// TIA Portal V20 export
// export: Created 2025-12-01T14:56:19.1379541Z, ExportSetting None, DisplayName Totally Integrated Automation Portal, DisplayVersion V20 Update 3, DisplayName TIA Portal Openness, DisplayVersion V20 Update 3, DisplayName TIA Portal Version Control Interface, DisplayVersion V20 Update 3, DisplayName STEP 7 Professional, DisplayVersion V20 Update 3, DisplayName STEP 7 Safety, DisplayVersion V20 Update 2, DisplayName WinCC Basic/Comfort/Advanced, DisplayVersion V20 Update 3, DisplayName WinCC Professional, DisplayVersion V20 Update 3, DisplayName WinCC Unified, DisplayVersion V20 Update 3
TYPE "i550 Estatus variador"
   STRUCT
      "Digital input 1" : Bool;   // DI1 Entrada digital 1 xxxx.0
      "Digital input 2" : Bool;   // DI2 Entrada digital 2 xxxx.1
      "Digital input 3" : Bool;   // DI3 Entrada digital 3 xxxx.2
      "Digital input 4" : Bool;   // DI4 Entrada digital 4 xxxx.3
      "Digital input 5" : Bool;   // DI5 Entrada digital 5 xxxx.4
      Running : Bool;
      "Release Holding Brake" : Bool;
      "Reserva 3" : Bool;
      "Ready for operation" : Bool;   // Dispositivo OK para su utilización
      "Auto setp active" : Bool;   // Modo auto activo
      "Actual speed = 0" : Bool;   // Velocidad actual = 0
      Error : Bool;   // Dispositivo en error
      "Safe torque off" : Bool;   // STO no activo en dispositivo
      "At current limit" : Bool;   // Corriente limite superada
      "At torque limit" : Bool;   // Par limite superado
      "Speed - set = act" : Bool;   // Consigna de velocidad alcanzada
   END_STRUCT;
END_TYPE
